VAR_GLOBAL CONSTANT

	nNumMaxMovers : UDINT :=10;
	nNumMaxTracks : UDINT :=3;
 	fMagnetEntry : LREAL := 10000;//8750; //PLEASE ENTER THE MAGNET ENTRY!!!
	fMagnetExit : LREAL := 10900; //PLEASE ENTER THE MAGNET EXIT!!!
END_VAR

VAR_GLOBAL
	aStopPositions : ARRAY [1..nNumMaxMovers] OF LREAL := [2400, 1700, 1000, 300];
	XtsOutterLoopOid: OTCID := 16#1010480;	
	XtsShortcutOid: OTCID := 16#1010490;
	
	MoverArrive : BOOL;
	MoverArrived : BOOL;
END_VAR

VAR_GLOBAL PERSISTENT
	nNumMovers: UDINT := 4;
	nMoverSartupPos : ARRAY[1..nNumMaxMovers] OF MoverSort;
END_VAR

(* stored: Version 1.1.0.1, ProductVersion 3.1.4024.12
   GVL GVL_General: Id {027beb7e-728e-4aeb-a930-890d17a65a81} *)
